FUNCTION_BLOCK E_SEL_STRING (* Event-driven STRING selection *)
  (* Standard: 61499-1; Classification: Math; Function: Event-driven selection *)
  (* Version 0.0, 2001-11-27, JHC, Rockwell Automation, Derived from E_SEL_WSTRING. *)
  (* Compiler header: package fb.rt.math; *)
  (* Compiler Java IBM VisualAge 3.0 *)
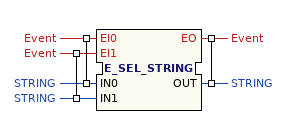
  EVENT_INPUT
    EI0 WITH IN0; (* Select INO *)
    EI1 WITH IN1; (* Select INO *)
  END_EVENT
  EVENT_OUTPUT
    EO WITH OUT; (* New selection event *)
  END_EVENT
  VAR_INPUT
    IN0 : STRING; (* Selected by EI0 *)
    IN1 : STRING; (* Selected by EI1 *)
  END_VAR
  VAR_OUTPUT
    OUT : STRING; (* Selected value *)
  END_VAR
END_FUNCTION_BLOCK
